// TIA Portal V16 export
// export: Created 2021-04-06T19:52:17.7285338Z, ExportSetting WithDefaults, DisplayName Totally Integrated Automation Portal, DisplayVersion V16, DisplayName TIA Portal Version Control Interface, DisplayVersion V16, DisplayName TIA Portal Openness, DisplayVersion V16, DisplayName STEP 7 Professional, DisplayVersion V16, DisplayName STEP 7 Safety, DisplayVersion V16, DisplayName WinCC Unified SCADA Engineering System, DisplayVersion V16
DATA_BLOCK "IO"   // DB10
{ S7_Optimized_Access := 'TRUE' }
VERSION : 0.1
// stored: AutoNumber false, DBAccessibleFromOPCUA true, IsOnlyStoredInLoadMemory false, IsRetainMemResEnabled false, IsWriteProtectedInAS false, MemoryReserve 100
   VAR
      input : Struct
         buttonControlCircuit : Bool;   // цепи управления
         buttonStart : Bool;   // Старт
         buttonStop : Bool;   // Стоп
         buttonAlarmStop : Bool;   // Аварийный стоп
         M_alarmCB : Array[0..2] of Bool;   // М - авария автоматического выключателя
         isNormalElectrical : Bool;   // Сеть в норме
         sensorOverflowReceiverTable : Bool;   // Датчик пересыпа приемного стола
         YP_ReadyAccept : Array[0..2] of Bool;   // УП - готов принять
         YP_StartDozing : Array[0..2] of Bool;   // УП - запуск дозирования
      END_STRUCT;
      output : Struct
         lampBlue : Bool;   // Синяя лампа
         lampGreen : Bool;   // Зеленая лампа
         lampRed : Bool;   // Красная лампа
         qOn_ControlCurcuit : Bool;   // включение цепей управления
         Yq_ReadyDoze : Array[0..2] of Bool;   // УП - доза готова
         Conv_FRV : Array[0..2] of Bool;   // Конвейер1 - вперед
         Conv_REV : Array[0..2] of Bool;   // Конвейер1 - назад
         Door_open : Array[0..12] of Bool;   // Лопатка - открыть
         Door_close : Array[0..12] of Bool;   // Лопатка - закрыть
         Bunker_leftOpen : Array[0..12] of Bool;   // Бункер - открыть влево
         Bunker_leftClose : Array[0..12] of Bool;   // Бункер - закрыть влево
         Bunker_rightOpen : Array[0..12] of Bool;   // Бункер - открыть вправо
         Bunker_rightClose : Array[0..12] of Bool;   // Бункер - закрыть вправо
         flipper_Up : Bool;   // управление плавником вверх
         flipper_Down : Bool;   // управление плавником вниз
         vibroTable : Array[0..2] of Bool;   // управление вибростолом
         vibroLot : Array[0..12] of Bool;   // управление вибролотком
         setVibration : Real;   // уставка вибрации
         setSpeed : Real;   // уставка скорости конвейера
         convSource : Bool;   // запуск питателя
      END_STRUCT;
   END_VAR
BEGIN
END_DATA_BLOCK
